FUNCTION "PE_W_Block1_old" : Void
{ S7_Optimized_Access := 'TRUE' }
VERSION : 0.1
   VAR_INPUT
      In_Data : "W_PE";   // pcs
   END_VAR

   VAR_OUTPUT
      Out_Data : Array[1..125] of Word;
   END_VAR


BEGIN
	REGION
	    #Out_Data[1] := INT_TO_WORD(#In_Data."iUserPswIns");
	END_REGION
END_FUNCTION

